// TIA Portal V18 export
DATA_BLOCK "BoilerAlarms"   // DB1015
{ S7_Optimized_Access := 'TRUE' }
VERSION : 0.1
// stored: AutoNumber false, DBAccessibleFromOPCUA true, IsOnlyStoredInLoadMemory false, IsRetainMemResEnabled false, IsWriteProtectedInAS false, MemoryReserve 100
   VAR
      Summary { S7_SetPoint := 'True'} : "UDT_BoilersSummaryAlarms";
   END_VAR
BEGIN
END_DATA_BLOCK
